FUNCTION_BLOCK PytorchHubModel
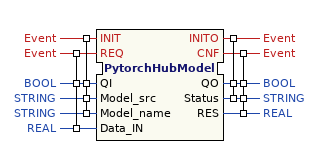
  EVENT_INPUT
    INIT WITH QI, Model_src, Model_name; (* Initialization Request *)
    REQ WITH QI, Data_IN; (* Normal Execution Request *)
  END_EVENT
  EVENT_OUTPUT
    INITO WITH QO, Status; (* Initialization Confirm *)
    CNF WITH QO, RES, Status; (* Execution Confirmation *)
  END_EVENT
  VAR_INPUT
    QI : BOOL; (* Input event qualifier *)
    Model_src : STRING;
    Model_name : STRING;
    Data_IN : REAL;
  END_VAR
  VAR_OUTPUT
    QO : BOOL; (* Output event qualifier *)
    Status : STRING;
    RES : REAL;
  END_VAR
END_FUNCTION_BLOCK
